// SIMATIC S7-200 project (STEP 7-Micro/WIN), CPU 224XP REL 02.01

SYMBOL_TABLE USUARIO1
up               I0.0     // ascendente
down             I0.1     // descender
reset            I0.2     // reset
bit_cero         Q0.0
bit_uno          Q0.1
bit_dos          Q0.2
bit_tres         Q0.3
bit_cuatro       Q0.4
bit_cinco        Q0.5
bit_seis         Q0.6
END_SYMBOL_TABLE

ORGANIZATION_BLOCK PRINCIPAL:OB1
TITLE=COMENTARIOS DEL PROGRAMA
BEGIN
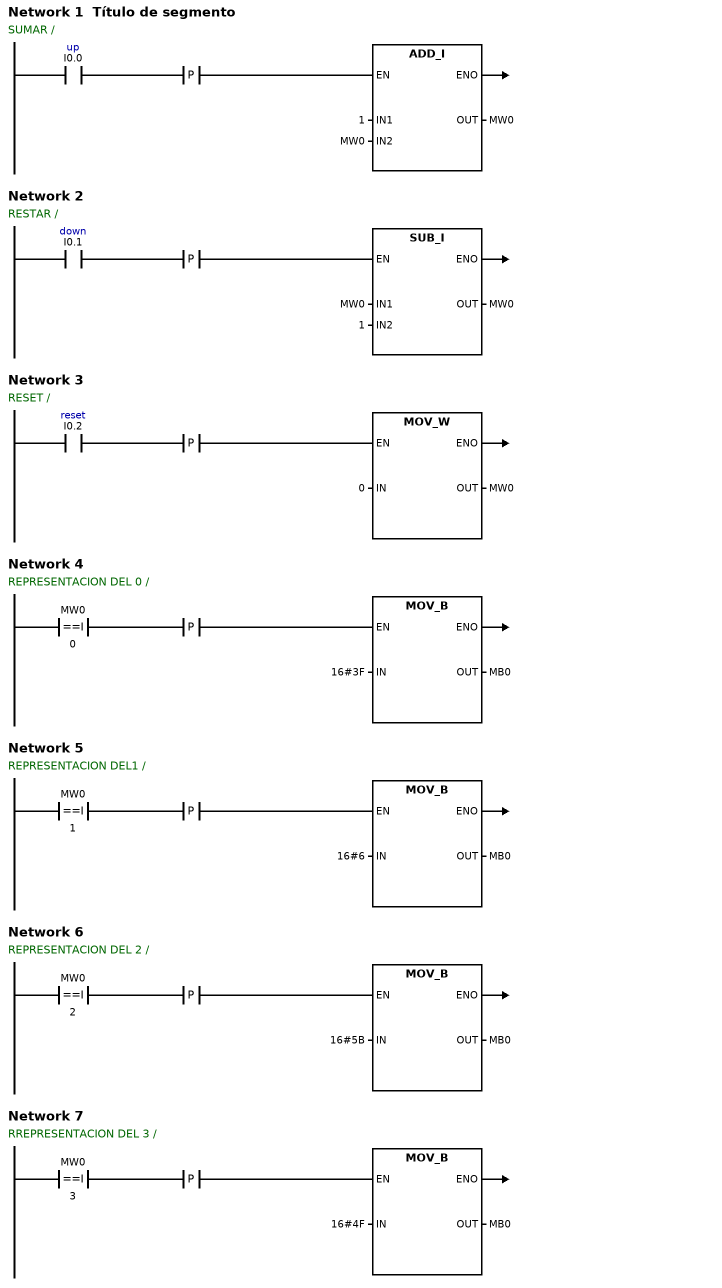
Network 1 // Título de segmento
// SUMAR
// 
LD     up:I0.0
EU
+I     1, MW0
Network 2
// RESTAR
// 
LD     down:I0.1
EU
-I     1, MW0
Network 3
// RESET
// 
LD     reset:I0.2
EU
MOVW   0, MW0
Network 4
// REPRESENTACION DEL 0
// 
LDW=   MW0, 0
EU
MOVB   16#3F, MB0
Network 5
// REPRESENTACION DEL1
// 
LDW=   MW0, 1
EU
MOVB   16#6, MB0
Network 6
// REPRESENTACION DEL 2
// 
LDW=   MW0, 2
EU
MOVB   16#5B, MB0
Network 7
// RREPRESENTACION DEL 3
// 
LDW=   MW0, 3
EU
MOVB   16#4F, MB0
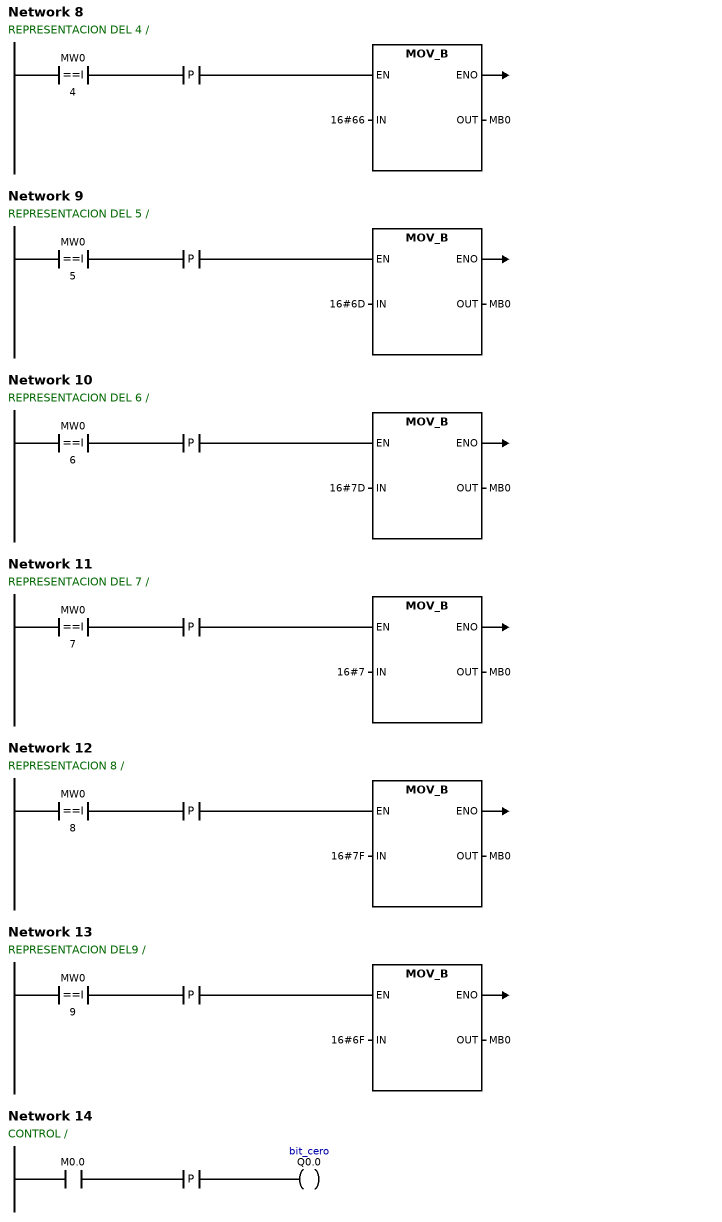
Network 8
// REPRESENTACION DEL 4
// 
LDW=   MW0, 4
EU
MOVB   16#66, MB0
Network 9
// REPRESENTACION DEL 5
// 
LDW=   MW0, 5
EU
MOVB   16#6D, MB0
Network 10
// REPRESENTACION DEL 6
// 
LDW=   MW0, 6
EU
MOVB   16#7D, MB0
Network 11
// REPRESENTACION DEL 7
// 
LDW=   MW0, 7
EU
MOVB   16#7, MB0
Network 12
// REPRESENTACION 8
// 
LDW=   MW0, 8
EU
MOVB   16#7F, MB0
Network 13
// REPRESENTACION DEL9
// 
LDW=   MW0, 9
EU
MOVB   16#6F, MB0
Network 14
// CONTROL
// 
LD     M0.0
EU
=      bit_cero:Q0.0
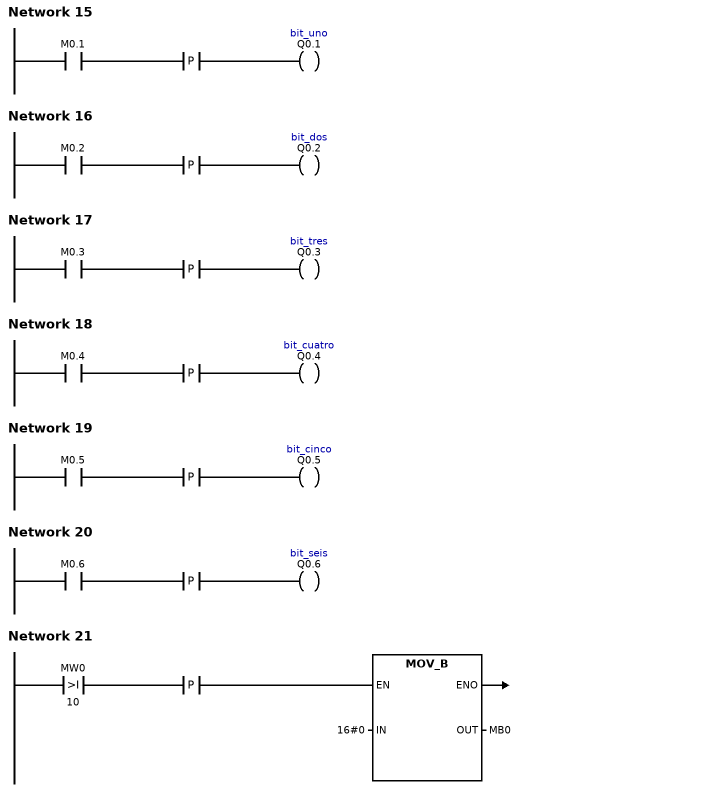
Network 15
LD     M0.1
EU
=      bit_uno:Q0.1
Network 16
LD     M0.2
EU
=      bit_dos:Q0.2
Network 17
LD     M0.3
EU
=      bit_tres:Q0.3
Network 18
LD     M0.4
EU
=      bit_cuatro:Q0.4
Network 19
LD     M0.5
EU
=      bit_cinco:Q0.5
Network 20
LD     M0.6
EU
=      bit_seis:Q0.6
Network 21
LDW>   MW0, 10
EU
MOVB   16#0, MB0
END_ORGANIZATION_BLOCK
